// TIA Portal V20 export
DATA_BLOCK "HmiInterface"   // DB96
// stored: Access Published, MemoryReserve 100, Namespace Unit1.Em5
   VAR
      em : "LAF_typeEmInterface";
      emHomedCheck : "Unit1.Em5.typeEmHomedCheck";
      cm : "Unit1.Em5.typeCmInterface";
      manualInput : "LER_typeSequenceInterface";
   END_VAR
   VAR RETAIN
      cmNgAndManualInputAxisY : "LBC_typeAxis64PosInterface";
      cmMagazineAxisZ : "LBC_typeAxis64PosInterface";
      cmNgAndManualInputCylinderUpDown : "LBC_typeTwoWayActuatorInterface";
      cmNgAndManualInputVacuum1OnOff : "LBC_typeTwoWayActuatorInterface";
      cmNgAndManualInputVacuum2OnOff : "LBC_typeTwoWayActuatorInterface";
      cmNgAndManualInputVibrator1OnOff : "LBC_typeTwoWayActuatorInterface";
      cmNgAndManualInputVibrator2OnOff : "LBC_typeTwoWayActuatorInterface";
      cmMagazineLockCylinderUpDown : "LBC_typeTwoWayActuatorInterface";
      cmNgAndManaulInputMagazineElectrodeDetectionSensor : "LBC_typeDigitalSignalInterface";
      cmNgAndManualInputMagazineDetectionSensor : "LBC_typeDigitalSignalInterface";
      cmNgAndManualInputMagazineFullSensor : "LBC_typeDigitalSignalInterface";
      cmNgAndManualInputElectrodeDetectionSensor : "LBC_typeDigitalSignalInterface";
      cmMagazineSafetyPinIdlePosition : "LBC_typeDigitalSignalInterface";
      cmNgAndManualInputAxisY_TorqueCal : "LER_typeServoTorqueCalInterface";
      cmMagazineAxisZ_TorqueCal : "LER_typeServoTorqueCalInterface";
   END_VAR
BEGIN
END_DATA_BLOCK
